FUNCTION_BLOCK FB_SingleDrive_Conveyor_With_Out_Sensor_And_Stopper EXTENDS FB_SingleDrive_Conveyor_With_Out_Sensor

VAR
END_VAR

END_FUNCTION_BLOCK

(* stored: Version 1.1.0.1, ProductVersion 3.1.4024.15
   POU FB_SingleDrive_Conveyor_With_Out_Sensor_And_Stopper: Id {58c91069-80ff-485d-ae0c-46ae716cb6b6}, SpecialFunc None *)
